TYPE st_Ledstrip_params :
STRUCT
	IP				: STRING 	:= '192.168.1.43'; //arduino controller only
	Numleds			: BYTE		:= 116;
	ColorOrder		: eColorOrder := eColorOrder.GRB;
END_STRUCT
END_TYPE

(* stored: Version 1.1.0.1, ProductVersion 3.1.4026.18
   DUT st_Ledstrip_params: Id {fc4d8e55-288c-49e2-a2e8-5db3d4238583} *)
